(* PLC project , Unknown 1 *)
(* stored: creationDateTime 2018-04-01T21:25:21, modificationDateTime 2018-05-24T16:45:06 *)

PROGRAM MAIN
  VAR_INPUT
    IN : INT;
  END_VAR
  VAR
    RET : INT;
  END_VAR
  VAR_OUTPUT
    OUT1 : INT;
  END_VAR

            RET := SFUN_SERVO_INPUT_UPDATE(0);
RET := SFUN_RCMODE_READ(0);

IF IN = 1 OR RET = 1 THEN
   RET := SFUN_SERVO_POWERON(1);
ELSE
   RET := SFUN_SERVO_POWEROFF(1);
   RET := SFUN_RCPLC_SERVOFLAG_SET(0);
END_IF;

IF RET = 1 THEN
   RET := SFUN_RCPLC_SERVOFLAG_SET(1);
   IF RET = 1 THEN
      RET := SFUN_INTERP_UPDATE(0);
      RET := SFUN_SERVO_OUTPUT_UPDATE(0);
   END_IF;
END_IF;
          
END_PROGRAM

CONFIGURATION config
  RESOURCE Resource1 ON PLC
    VAR_GLOBAL
      W : BYTE;
    END_VAR
    TASK fast(INTERVAL := T#8ms, PRIORITY := 90);
    PROGRAM P1 WITH fast : MAIN;
  END_RESOURCE
END_CONFIGURATION
